// TwinCAT 3 PLC project Untitled1
// ProgramVersion: 3.1.4024.0
// libraries:
//   Tc2_Standard, * (Beckhoff Automation GmbH)
//   Tc2_System, * (Beckhoff Automation GmbH)
//   Tc2_Utilities, * (Beckhoff Automation GmbH)
//   Tc3_Module, * (Beckhoff Automation GmbH)
// project tree:
//   / PlcTask.TcTTO
//   POUs/ MAIN.TcPOU
// real-time tasks:
//   TASK PlcTask: cycle T#10ms, priority 20, ADS port 350

CONFIGURATION Untitled1
    RESOURCE PLC ON TwinCAT3
        TASK PlcTask(INTERVAL := T#10ms, PRIORITY := 20);
        PROGRAM MAIN WITH PlcTask : MAIN;
    END_RESOURCE
END_CONFIGURATION

// ---- POUs/MAIN.TcPOU
PROGRAM MAIN
VAR
//Declare the two strings which are going to exceed the limit of 255 characters when concatenated 
string1 : STRING(1000) := 'Lorem ipsum odor amet, consectetuer adipiscing elit. Non per dapis himenaeos eros justo consectetur nam. Lorem ipsum odor amet, consectetuer adipiscing elit. Faucibus nec a Test Lorem ipsum odor amet, consectetuer adipiscing elit. Faucibus nec a Test';
string2 : STRING(1000) := 'Lorem ipsum odor amet, consectetuer adipiscing elit. Faucibus nec a Test Lorem ipsum odor amet, consectetuer adipiscing elit. Faucibus nec a Test Lorem ipsum odor amet, consectetuer adipiscing elit. Faucibus nec a Test Lorem ipsum odor amet, consectetuer adipiscing elit. Faucibus nec a Test';
//Declare a 3rd string for the concatenated result to be stored and set it to the desired size.
string3 : STRING(1000);


//Declare 3 string pointers 
pString1 : POINTER TO STRING;
pString2 : POINTER TO STRING;
pString3 : POINTER TO STRING;


END_VAR

//assign each string pointer variable to the value of each string 
pString1 := ADR(string1);
pString2 := ADR(string2);
pString3 := ADR(string3);

concat2(pString1, pString2, pString3, 1000);

END_PROGRAM
